TYPE ST_Filter_Current_Hexapod_Robot_Output :
STRUCT
	Current_Monitor: matrix_18_real_T;
END_STRUCT
END_TYPE

(* stored: Version 1.1.0.1, ProductVersion 3.1.4020.12
   DUT ST_Filter_Current_Hexapod_Robot_Output: Id {2230971b-360c-4c95-a302-0e09ae5312e7} *)
